// Mitsubishi GX Works2 project: PART_REPEAT_SEQUENCE2   PLC: Q03UDV

PROGRAM MAIN
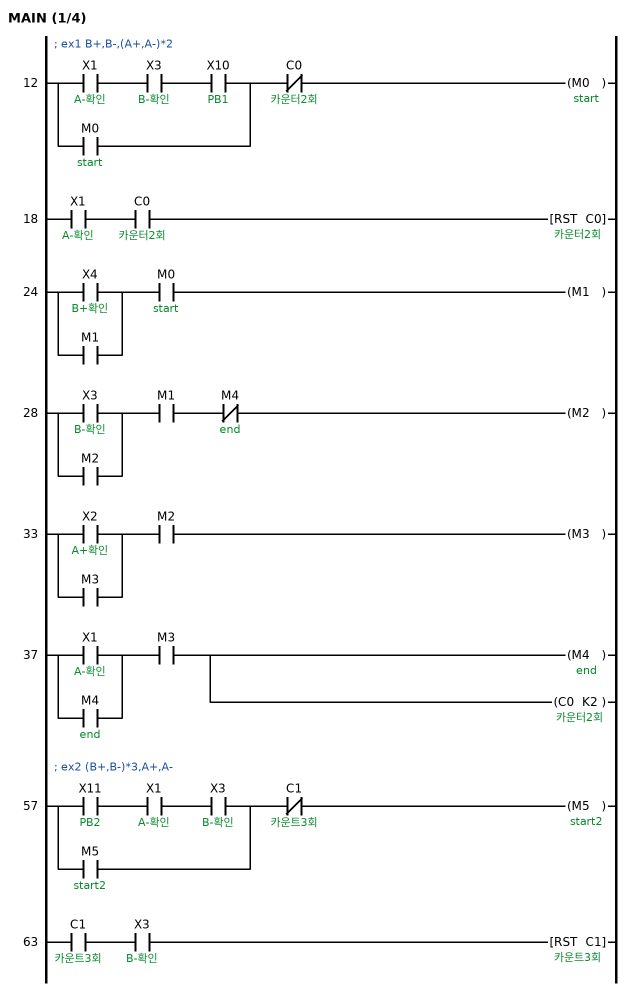
; ex1 B+,B-,(A+,A-)*2
12    LD      X1  ; A-확인
      AND     X3  ; B-확인
      AND     X10  ; PB1
      OR      M0  ; start
      ANI     C0  ; 카운터2회
      OUT     M0  ; start
18    LD      X1  ; A-확인
      AND     C0  ; 카운터2회
      RST     C0  ; 카운터2회
24    LD      X4  ; B+확인
      OR      M1
      AND     M0  ; start
      OUT     M1
28    LD      X3  ; B-확인
      OR      M2
      AND     M1
      ANI     M4  ; end
      OUT     M2
33    LD      X2  ; A+확인
      OR      M3
      AND     M2
      OUT     M3
37    LD      X1  ; A-확인
      OR      M4  ; end
      AND     M3
      OUT     M4  ; end
      OUT     C0 K2  ; 카운터2회
; ex2 (B+,B-)*3,A+,A-
57    LD      X11  ; PB2
      AND     X1  ; A-확인
      AND     X3  ; B-확인
      OR      M5  ; start2
      ANI     C1  ; 카운트3회
      OUT     M5  ; start2
63    LD      C1  ; 카운트3회
      AND     X3  ; B-확인
      RST     C1  ; 카운트3회
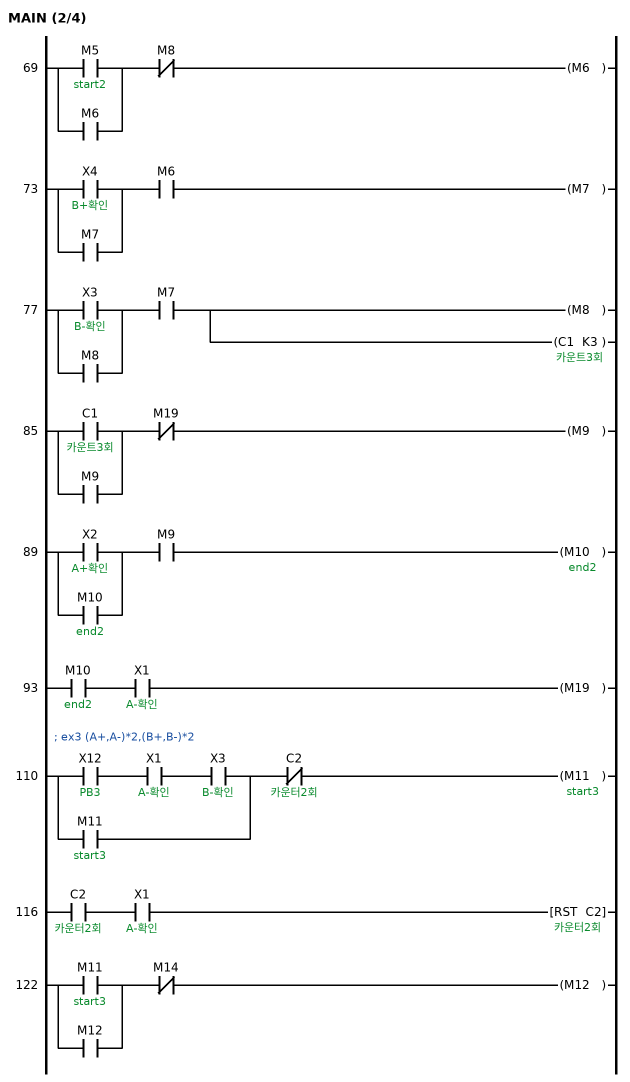
69    LD      M5  ; start2
      OR      M6
      ANI     M8
      OUT     M6
73    LD      X4  ; B+확인
      OR      M7
      AND     M6
      OUT     M7
77    LD      X3  ; B-확인
      OR      M8
      AND     M7
      OUT     M8
      OUT     C1 K3  ; 카운트3회
85    LD      C1  ; 카운트3회
      OR      M9
      ANI     M19
      OUT     M9
89    LD      X2  ; A+확인
      OR      M10  ; end2
      AND     M9
      OUT     M10  ; end2
93    LD      M10  ; end2
      AND     X1  ; A-확인
      OUT     M19
; ex3 (A+,A-)*2,(B+,B-)*2
110   LD      X12  ; PB3
      AND     X1  ; A-확인
      AND     X3  ; B-확인
      OR      M11  ; start3
      ANI     C2  ; 카운터2회
      OUT     M11  ; start3
116   LD      C2  ; 카운터2회
      AND     X1  ; A-확인
      RST     C2  ; 카운터2회
122   LD      M11  ; start3
      OR      M12
      ANI     M14
      OUT     M12
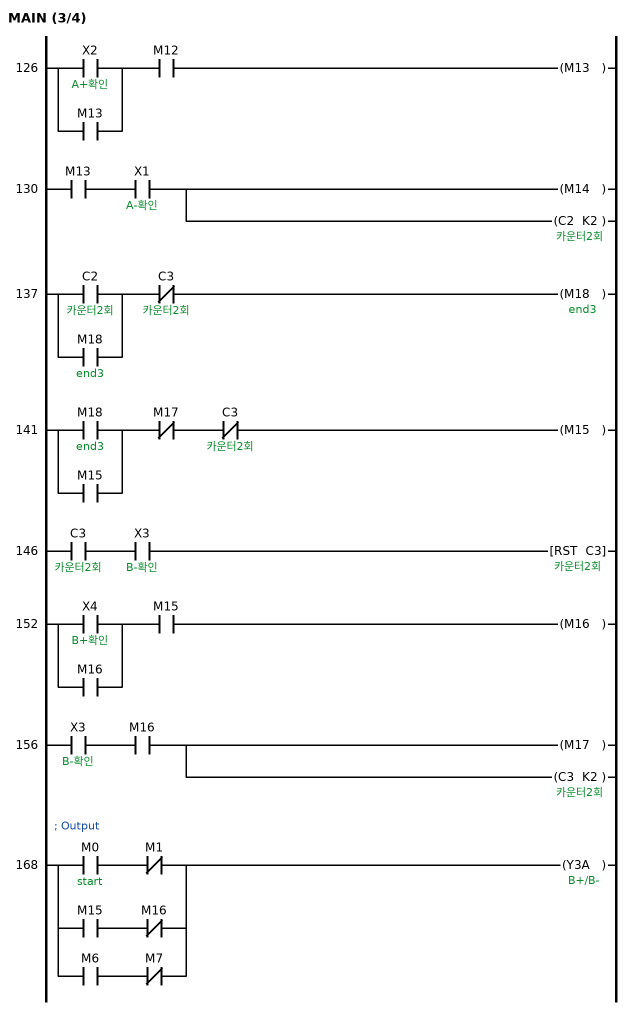
126   LD      X2  ; A+확인
      OR      M13
      AND     M12
      OUT     M13
130   LD      M13
      AND     X1  ; A-확인
      OUT     M14
      OUT     C2 K2  ; 카운터2회
137   LD      C2  ; 카운터2회
      OR      M18  ; end3
      ANI     C3  ; 카운터2회
      OUT     M18  ; end3
141   LD      M18  ; end3
      OR      M15
      ANI     M17
      ANI     C3  ; 카운터2회
      OUT     M15
146   LD      C3  ; 카운터2회
      AND     X3  ; B-확인
      RST     C3  ; 카운터2회
152   LD      X4  ; B+확인
      OR      M16
      AND     M15
      OUT     M16
156   LD      X3  ; B-확인
      AND     M16
      OUT     M17
      OUT     C3 K2  ; 카운터2회
; Output
168   LD      M0  ; start
      ANI     M1
      LD      M15
      ANI     M16
      ORB
      LD      M6
      ANI     M7
      ORB
      OUT     Y3A  ; B+/B-
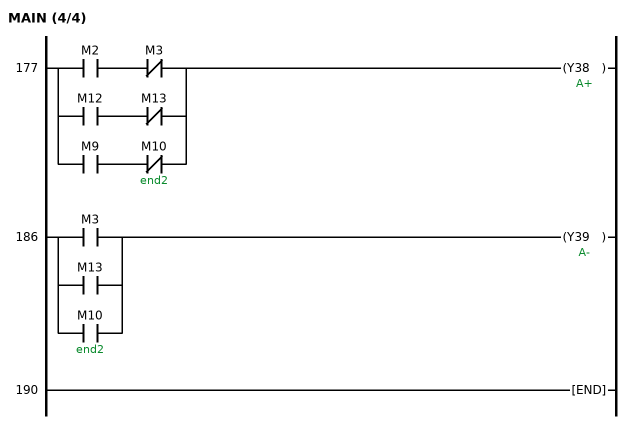
177   LD      M2
      ANI     M3
      LD      M12
      ANI     M13
      ORB
      LD      M9
      ANI     M10  ; end2
      ORB
      OUT     Y38  ; A+
186   LD      M3
      OR      M13
      OR      M10  ; end2
      OUT     Y39  ; A-
190   END
END_PROGRAM
